TYPE test :
STRUCT
	Id: LINT;
	Sync: BOOL;
	Vari: REAL;
	//Timestamp: DT;
END_STRUCT
END_TYPE

(* stored: Version 1.1.0.1, ProductVersion 3.1.4024.4
   DUT test: Id {a041a85b-a0d7-4bb7-a219-415fa1a914fe} *)
